{attribute 'qualified_only'}
{attribute 'strict'}
{attribute 'to_string'}
TYPE DUT_Command_PositionType :
(
	AbsolutePosition := 0,
	RelativePosition := 1
);
END_TYPE

(* stored: Version 1.1.0.1
   EnumerationTextList DUT_Command_PositionType: Id {cafbdcf3-c8c4-4c4d-b394-6a0cfd8bc796} *)
